FUNCTION IncINT : INT				// Increments the given UINT value
VAR_IN_OUT
	ioNum:	INT;		// Value to increment
END_VAR

IncINT := ioNum := ioNum + 1;

END_FUNCTION

(* stored: Version 1.1.0.1, ProductVersion 3.1.4026.18
   POU IncINT: Id {7b95fc8e-a3f0-4c3d-b28a-468cad96c581}, SpecialFunc None *)
